INTERFACE I_Logger EXTENDS I_FileAccess

METHOD LogError
VAR_INPUT
END_VAR
END_METHOD

METHOD LogGeneric
VAR_INPUT
END_VAR
END_METHOD

METHOD LogInfo
VAR_INPUT
END_VAR
END_METHOD

METHOD LogWarning
VAR_INPUT
END_VAR
END_METHOD

END_INTERFACE

(* stored: Version 1.1.0.1, ProductVersion 3.1.4024.13
   Itf I_Logger: Id {0db69b78-3cea-0d64-1476-a39aaa2ee03e}
   Method LogError: Id {df7195e3-abce-008e-317c-131e25ddee27}
   Method LogGeneric: Id {77fea8d6-3bb9-07fa-3ca3-4cc1f73392ba}
   Method LogInfo: Id {7f5adfde-a437-082b-0720-4b9797ec4c1e}
   Method LogWarning: Id {34db8310-88e2-0df4-13c7-08648a8d84fc} *)
